  PROC DrawPart12()
    MoveL Offs(pOrigin,202.25,-93.12,-6.00),v60,z5,tcp\WObj:=Plywood;
    MoveL Offs(pOrigin,203.00,-90.38,-6.00),vTravel,z5,tcp\WObj:=Plywood;
    MoveL Offs(pOrigin,203.00,-90.38,-0.00),v60,z0,tcp\WObj:=Plywood;
    MoveL Offs(pOrigin,202.80,-90.22,-0.00),v40,z0,tcp\WObj:=Plywood;
    MoveL Offs(pOrigin,203.15,-89.57,-0.00),v40,z0,tcp\WObj:=Plywood;
    MoveL Offs(pOrigin,202.30,-90.18,-0.00),v40,z0,tcp\WObj:=Plywood;
    MoveL Offs(pOrigin,202.25,-88.72,-0.00),v40,z0,tcp\WObj:=Plywood;
    MoveL Offs(pOrigin,202.60,-88.12,-0.00),v40,z0,tcp\WObj:=Plywood;
    MoveL Offs(pOrigin,202.25,-87.82,-0.00),v40,z0,tcp\WObj:=Plywood;
    MoveL Offs(pOrigin,202.25,-72.22,-0.00),v40,z0,tcp\WObj:=Plywood;
    MoveL Offs(pOrigin,204.35,-70.43,-0.00),v40,z0,tcp\WObj:=Plywood;
    MoveL Offs(pOrigin,203.30,-69.22,-0.00),v40,z0,tcp\WObj:=Plywood;
    MoveL Offs(pOrigin,202.25,-68.93,-0.00),v40,z0,tcp\WObj:=Plywood;
    MoveL Offs(pOrigin,202.10,-50.83,-0.00),v40,z0,tcp\WObj:=Plywood;
    MoveL Offs(pOrigin,210.05,-50.92,-0.00),v40,z0,tcp\WObj:=Plywood;
    MoveL Offs(pOrigin,214.70,-52.12,-0.00),v40,z0,tcp\WObj:=Plywood;
    MoveL Offs(pOrigin,217.55,-53.28,-0.00),v40,z0,tcp\WObj:=Plywood;
    MoveL Offs(pOrigin,222.65,-56.47,-0.00),v40,z0,tcp\WObj:=Plywood;
    MoveL Offs(pOrigin,225.65,-59.33,-0.00),v40,z0,tcp\WObj:=Plywood;
    MoveL Offs(pOrigin,227.75,-62.03,-0.00),v40,z0,tcp\WObj:=Plywood;
    MoveL Offs(pOrigin,229.80,-65.62,-0.00),v40,z0,tcp\WObj:=Plywood;
    MoveL Offs(pOrigin,231.05,-68.78,-0.00),v40,z0,tcp\WObj:=Plywood;
    MoveL Offs(pOrigin,232.25,-74.18,-0.00),v40,z0,tcp\WObj:=Plywood;
    MoveL Offs(pOrigin,232.40,-76.88,-0.00),v40,z0,tcp\WObj:=Plywood;
    MoveL Offs(pOrigin,232.25,-80.93,-0.00),v40,z0,tcp\WObj:=Plywood;
    MoveL Offs(pOrigin,231.50,-84.68,-0.00),v40,z0,tcp\WObj:=Plywood;
    MoveL Offs(pOrigin,230.20,-88.28,-0.00),v40,z0,tcp\WObj:=Plywood;
    MoveL Offs(pOrigin,228.95,-90.38,-0.00),v40,z0,tcp\WObj:=Plywood;
    MoveL Offs(pOrigin,203.00,-90.38,-0.00),v40,z0,tcp\WObj:=Plywood;
    MoveL Offs(pOrigin,203.45,-89.47,-0.00),v40,z0,tcp\WObj:=Plywood;
    MoveL Offs(pOrigin,203.90,-89.32,-0.00),v40,z0,tcp\WObj:=Plywood;
    MoveL Offs(pOrigin,203.45,-88.88,-0.00),v40,z0,tcp\WObj:=Plywood;
    MoveL Offs(pOrigin,203.45,-89.47,-0.00),v40,z0,tcp\WObj:=Plywood;
    MoveL Offs(pOrigin,203.90,-89.18,-0.00),v40,z0,tcp\WObj:=Plywood;
    MoveL Offs(pOrigin,203.60,-88.88,-0.00),v40,z0,tcp\WObj:=Plywood;
    MoveL Offs(pOrigin,203.30,-89.03,-0.00),v40,z0,tcp\WObj:=Plywood;
    MoveL Offs(pOrigin,203.45,-89.47,-0.00),v40,fine,tcp\WObj:=Plywood;
    MoveL Offs(pOrigin,203.45,-89.47,-6.00),v60,z5,tcp\WObj:=Plywood;
    MoveL Offs(pOrigin,198.50,-85.88,-6.00),vTravel,z5,tcp\WObj:=Plywood;
    MoveL Offs(pOrigin,198.50,-85.88,-0.00),v60,z0,tcp\WObj:=Plywood;
    MoveL Offs(pOrigin,198.20,-85.57,-0.00),v40,z0,tcp\WObj:=Plywood;
    MoveL Offs(pOrigin,197.75,-85.88,-0.00),v40,z0,tcp\WObj:=Plywood;
    MoveL Offs(pOrigin,198.35,-86.03,-0.00),v40,z0,tcp\WObj:=Plywood;
    MoveL Offs(pOrigin,198.20,-85.57,-0.00),v40,z0,tcp\WObj:=Plywood;
    MoveL Offs(pOrigin,197.75,-85.88,-0.00),v40,z0,tcp\WObj:=Plywood;
    MoveL Offs(pOrigin,198.50,-85.88,-0.00),v40,z0,tcp\WObj:=Plywood;
    MoveL Offs(pOrigin,197.60,-85.12,-0.00),v40,z0,tcp\WObj:=Plywood;
    MoveL Offs(pOrigin,197.45,-84.32,-0.00),v40,z0,tcp\WObj:=Plywood;
    MoveL Offs(pOrigin,197.15,-84.68,-0.00),v40,z0,tcp\WObj:=Plywood;
    MoveL Offs(pOrigin,197.30,-85.38,-0.00),v40,z0,tcp\WObj:=Plywood;
    MoveL Offs(pOrigin,197.60,-85.12,-0.00),v40,z0,tcp\WObj:=Plywood;
    MoveL Offs(pOrigin,197.65,-84.22,-0.00),v40,z0,tcp\WObj:=Plywood;
    MoveL Offs(pOrigin,199.00,-83.93,-0.00),v40,z0,tcp\WObj:=Plywood;
    MoveL Offs(pOrigin,198.35,-83.53,-0.00),v40,z0,tcp\WObj:=Plywood;
    MoveL Offs(pOrigin,197.65,-84.22,-0.00),v40,fine,tcp\WObj:=Plywood;
    MoveL Offs(pOrigin,197.65,-84.22,-6.00),v60,z5,tcp\WObj:=Plywood;
    MoveL Offs(pOrigin,197.30,-79.53,-6.00),vTravel,z5,tcp\WObj:=Plywood;
    MoveL Offs(pOrigin,197.30,-79.53,-0.00),v60,z0,tcp\WObj:=Plywood;
    MoveL Offs(pOrigin,198.80,-78.38,-0.00),v40,z0,tcp\WObj:=Plywood;
    MoveL Offs(pOrigin,199.10,-77.78,-0.00),v40,z0,tcp\WObj:=Plywood;
    MoveL Offs(pOrigin,199.05,-76.72,-0.00),v40,z0,tcp\WObj:=Plywood;
    MoveL Offs(pOrigin,197.90,-75.82,-0.00),v40,z0,tcp\WObj:=Plywood;
    MoveL Offs(pOrigin,197.50,-76.28,-0.00),v40,z0,tcp\WObj:=Plywood;
    MoveL Offs(pOrigin,198.40,-76.88,-0.00),v40,z0,tcp\WObj:=Plywood;
    MoveL Offs(pOrigin,198.50,-77.32,-0.00),v40,z0,tcp\WObj:=Plywood;
    MoveL Offs(pOrigin,197.15,-76.57,-0.00),v40,z0,tcp\WObj:=Plywood;
    MoveL Offs(pOrigin,196.40,-77.03,-0.00),v40,z0,tcp\WObj:=Plywood;
    MoveL Offs(pOrigin,195.80,-77.93,-0.00),v40,z0,tcp\WObj:=Plywood;
    MoveL Offs(pOrigin,195.90,-78.68,-0.00),v40,z0,tcp\WObj:=Plywood;
    MoveL Offs(pOrigin,196.85,-79.53,-0.00),v40,z0,tcp\WObj:=Plywood;
    MoveL Offs(pOrigin,197.30,-79.53,-0.00),v40,z0,tcp\WObj:=Plywood;
    MoveL Offs(pOrigin,196.85,-78.78,-0.00),v40,z0,tcp\WObj:=Plywood;
    MoveL Offs(pOrigin,196.65,-77.93,-0.00),v40,z0,tcp\WObj:=Plywood;
    MoveL Offs(pOrigin,197.45,-77.38,-0.00),v40,z0,tcp\WObj:=Plywood;
    MoveL Offs(pOrigin,197.65,-78.22,-0.00),v40,z0,tcp\WObj:=Plywood;
    MoveL Offs(pOrigin,196.85,-78.78,-0.00),v40,fine,tcp\WObj:=Plywood;
    MoveL Offs(pOrigin,196.85,-78.78,-6.00),v60,z5,tcp\WObj:=Plywood;
    MoveL Offs(pOrigin,195.80,-77.32,-6.00),vTravel,z5,tcp\WObj:=Plywood;
    MoveL Offs(pOrigin,195.80,-77.32,-0.00),v60,z0,tcp\WObj:=Plywood;
    MoveL Offs(pOrigin,196.90,-75.97,-0.00),v40,z0,tcp\WObj:=Plywood;
    MoveL Offs(pOrigin,196.55,-75.68,-0.00),v40,z0,tcp\WObj:=Plywood;
    MoveL Offs(pOrigin,195.35,-76.72,-0.00),v40,z0,tcp\WObj:=Plywood;
    MoveL Offs(pOrigin,194.80,-76.57,-0.00),v40,z0,tcp\WObj:=Plywood;
    MoveL Offs(pOrigin,194.80,-76.12,-0.00),v40,z0,tcp\WObj:=Plywood;
    MoveL Offs(pOrigin,195.95,-74.78,-0.00),v40,z0,tcp\WObj:=Plywood;
    MoveL Offs(pOrigin,195.65,-74.43,-0.00),v40,z0,tcp\WObj:=Plywood;
    MoveL Offs(pOrigin,194.90,-74.62,-0.00),v40,z0,tcp\WObj:=Plywood;
    MoveL Offs(pOrigin,195.00,-73.88,-0.00),v40,z0,tcp\WObj:=Plywood;
    MoveL Offs(pOrigin,194.35,-73.12,-0.00),v40,z0,tcp\WObj:=Plywood;
    MoveL Offs(pOrigin,194.60,-72.07,-0.00),v40,z0,tcp\WObj:=Plywood;
    MoveL Offs(pOrigin,194.15,-71.82,-0.00),v40,z0,tcp\WObj:=Plywood;
    MoveL Offs(pOrigin,192.85,-73.07,-0.00),v40,z0,tcp\WObj:=Plywood;
    MoveL Offs(pOrigin,193.30,-72.22,-0.00),v40,z0,tcp\WObj:=Plywood;
    MoveL Offs(pOrigin,192.80,-71.93,-0.00),v40,z0,tcp\WObj:=Plywood;
    MoveL Offs(pOrigin,191.45,-72.97,-0.00),v40,z0,tcp\WObj:=Plywood;
    MoveL Offs(pOrigin,191.25,-72.22,-0.00),v40,z0,tcp\WObj:=Plywood;
    MoveL Offs(pOrigin,192.20,-71.03,-0.00),v40,z0,tcp\WObj:=Plywood;
    MoveL Offs(pOrigin,191.75,-70.72,-0.00),v40,z0,tcp\WObj:=Plywood;
    MoveL Offs(pOrigin,191.00,-71.07,-0.00),v40,z0,tcp\WObj:=Plywood;
    MoveL Offs(pOrigin,189.85,-72.38,-0.00),v40,z0,tcp\WObj:=Plywood;
    MoveL Offs(pOrigin,189.95,-72.82,-0.00),v40,z0,tcp\WObj:=Plywood;
    MoveL Offs(pOrigin,191.00,-73.88,-0.00),v40,z0,tcp\WObj:=Plywood;
    MoveL Offs(pOrigin,191.75,-73.88,-0.00),v40,z0,tcp\WObj:=Plywood;
    MoveL Offs(pOrigin,192.35,-73.43,-0.00),v40,z0,tcp\WObj:=Plywood;
    MoveL Offs(pOrigin,191.75,-74.47,-0.00),v40,z0,tcp\WObj:=Plywood;
    MoveL Offs(pOrigin,192.50,-75.53,-0.00),v40,z0,tcp\WObj:=Plywood;
    MoveL Offs(pOrigin,193.95,-75.72,-0.00),v40,z0,tcp\WObj:=Plywood;
    MoveL Offs(pOrigin,193.75,-76.43,-0.00),v40,z0,tcp\WObj:=Plywood;
    MoveL Offs(pOrigin,194.75,-77.57,-0.00),v40,z0,tcp\WObj:=Plywood;
    MoveL Offs(pOrigin,195.80,-77.32,-0.00),v40,fine,tcp\WObj:=Plywood;
    MoveL Offs(pOrigin,195.80,-77.32,-6.00),v60,z5,tcp\WObj:=Plywood;
    MoveL Offs(pOrigin,193.85,-74.72,-6.00),vTravel,z5,tcp\WObj:=Plywood;
    MoveL Offs(pOrigin,193.85,-74.72,-0.00),v60,z0,tcp\WObj:=Plywood;
    MoveL Offs(pOrigin,193.00,-74.78,-0.00),v40,z0,tcp\WObj:=Plywood;
    MoveL Offs(pOrigin,193.25,-74.03,-0.00),v40,z0,tcp\WObj:=Plywood;
    MoveL Offs(pOrigin,194.00,-73.88,-0.00),v40,z0,tcp\WObj:=Plywood;
    MoveL Offs(pOrigin,193.85,-74.72,-0.00),v40,fine,tcp\WObj:=Plywood;
    MoveL Offs(pOrigin,193.85,-74.72,-6.00),v60,z5,tcp\WObj:=Plywood;
    MoveL Offs(pOrigin,191.40,-70.57,-6.00),vTravel,z5,tcp\WObj:=Plywood;
    MoveL Offs(pOrigin,191.40,-70.57,-0.00),v60,z0,tcp\WObj:=Plywood;
  ENDPROC

  PROC DrawPart13()
    MoveL Offs(pOrigin,190.55,-69.38,-0.00),v40,z0,tcp\WObj:=Plywood;
    MoveL Offs(pOrigin,189.80,-68.93,-0.00),v40,z0,tcp\WObj:=Plywood;
    MoveL Offs(pOrigin,188.95,-69.68,-0.00),v40,z0,tcp\WObj:=Plywood;
    MoveL Offs(pOrigin,189.45,-71.12,-0.00),v40,z0,tcp\WObj:=Plywood;
    MoveL Offs(pOrigin,188.75,-70.18,-0.00),v40,z0,tcp\WObj:=Plywood;
    MoveL Offs(pOrigin,188.30,-70.43,-0.00),v40,z0,tcp\WObj:=Plywood;
    MoveL Offs(pOrigin,188.60,-71.47,-0.00),v40,z0,tcp\WObj:=Plywood;
    MoveL Offs(pOrigin,189.35,-71.93,-0.00),v40,z0,tcp\WObj:=Plywood;
    MoveL Offs(pOrigin,189.95,-71.88,-0.00),v40,z0,tcp\WObj:=Plywood;
    MoveL Offs(pOrigin,191.40,-70.57,-0.00),v40,fine,tcp\WObj:=Plywood;
    MoveL Offs(pOrigin,191.40,-70.57,-6.00),v60,z5,tcp\WObj:=Plywood;
    MoveL Offs(pOrigin,190.10,-70.43,-6.00),vTravel,z5,tcp\WObj:=Plywood;
    MoveL Offs(pOrigin,190.10,-70.43,-0.00),v60,z0,tcp\WObj:=Plywood;
    MoveL Offs(pOrigin,189.80,-69.82,-0.00),v40,z0,tcp\WObj:=Plywood;
    MoveL Offs(pOrigin,190.10,-70.43,-0.00),v40,fine,tcp\WObj:=Plywood;
    MoveL Offs(pOrigin,190.10,-70.43,-6.00),v60,z5,tcp\WObj:=Plywood;
    MoveL Offs(pOrigin,188.65,-69.38,-6.00),vTravel,z5,tcp\WObj:=Plywood;
    MoveL Offs(pOrigin,188.65,-69.38,-0.00),v60,z0,tcp\WObj:=Plywood;
    MoveL Offs(pOrigin,187.70,-67.93,-0.00),v40,z0,tcp\WObj:=Plywood;
    MoveL Offs(pOrigin,188.45,-68.18,-0.00),v40,z0,tcp\WObj:=Plywood;
    MoveL Offs(pOrigin,188.75,-69.03,-0.00),v40,z0,tcp\WObj:=Plywood;
    MoveL Offs(pOrigin,189.15,-68.78,-0.00),v40,z0,tcp\WObj:=Plywood;
    MoveL Offs(pOrigin,189.10,-68.18,-0.00),v40,z0,tcp\WObj:=Plywood;
    MoveL Offs(pOrigin,188.45,-67.47,-0.00),v40,z0,tcp\WObj:=Plywood;
    MoveL Offs(pOrigin,187.40,-67.47,-0.00),v40,z0,tcp\WObj:=Plywood;
    MoveL Offs(pOrigin,186.70,-68.18,-0.00),v40,z0,tcp\WObj:=Plywood;
    MoveL Offs(pOrigin,186.50,-68.78,-0.00),v40,z0,tcp\WObj:=Plywood;
    MoveL Offs(pOrigin,187.25,-69.93,-0.00),v40,z0,tcp\WObj:=Plywood;
    MoveL Offs(pOrigin,188.15,-69.88,-0.00),v40,z0,tcp\WObj:=Plywood;
    MoveL Offs(pOrigin,188.65,-69.38,-0.00),v40,z0,tcp\WObj:=Plywood;
    MoveL Offs(pOrigin,187.80,-69.22,-0.00),v40,z0,tcp\WObj:=Plywood;
    MoveL Offs(pOrigin,187.25,-69.18,-0.00),v40,z0,tcp\WObj:=Plywood;
    MoveL Offs(pOrigin,187.15,-68.68,-0.00),v40,z0,tcp\WObj:=Plywood;
    MoveL Offs(pOrigin,187.80,-69.22,-0.00),v40,fine,tcp\WObj:=Plywood;
    MoveL Offs(pOrigin,187.80,-69.22,-6.00),v60,z5,tcp\WObj:=Plywood;
    MoveL Offs(pOrigin,186.45,-67.88,-6.00),vTravel,z5,tcp\WObj:=Plywood;
    MoveL Offs(pOrigin,186.45,-67.88,-0.00),v60,z0,tcp\WObj:=Plywood;
    MoveL Offs(pOrigin,187.35,-66.82,-0.00),v40,z0,tcp\WObj:=Plywood;
    MoveL Offs(pOrigin,187.25,-66.57,-0.00),v40,z0,tcp\WObj:=Plywood;
    MoveL Offs(pOrigin,185.45,-68.18,-0.00),v40,z0,tcp\WObj:=Plywood;
    MoveL Offs(pOrigin,185.20,-68.78,-0.00),v40,z0,tcp\WObj:=Plywood;
    MoveL Offs(pOrigin,186.45,-67.88,-0.00),v40,fine,tcp\WObj:=Plywood;
    MoveL Offs(pOrigin,186.45,-67.88,-6.00),v60,z5,tcp\WObj:=Plywood;
    MoveL Offs(pOrigin,186.50,-66.38,-6.00),vTravel,z5,tcp\WObj:=Plywood;
    MoveL Offs(pOrigin,186.50,-66.38,-0.00),v60,z0,tcp\WObj:=Plywood;
    MoveL Offs(pOrigin,186.50,-65.62,-0.00),v40,z0,tcp\WObj:=Plywood;
    MoveL Offs(pOrigin,186.50,-66.38,-0.00),v40,fine,tcp\WObj:=Plywood;
    MoveL Offs(pOrigin,186.50,-66.38,-6.00),v60,z5,tcp\WObj:=Plywood;
    MoveL Offs(pOrigin,185.30,-76.07,-6.00),vTravel,z5,tcp\WObj:=Plywood;
    MoveL Offs(pOrigin,185.30,-76.07,-0.00),v60,z0,tcp\WObj:=Plywood;
    MoveL Offs(pOrigin,185.05,-76.28,-0.00),v40,z0,tcp\WObj:=Plywood;
    MoveL Offs(pOrigin,185.75,-77.32,-0.00),v40,z0,tcp\WObj:=Plywood;
    MoveL Offs(pOrigin,185.05,-77.47,-0.00),v40,z0,tcp\WObj:=Plywood;
    MoveL Offs(pOrigin,185.00,-78.62,-0.00),v40,z0,tcp\WObj:=Plywood;
    MoveL Offs(pOrigin,186.25,-77.32,-0.00),v40,z0,tcp\WObj:=Plywood;
    MoveL Offs(pOrigin,185.30,-76.07,-0.00),v40,fine,tcp\WObj:=Plywood;
    MoveL Offs(pOrigin,185.30,-76.07,-6.00),v60,z5,tcp\WObj:=Plywood;
    MoveL Offs(pOrigin,184.05,-77.03,-6.00),vTravel,z5,tcp\WObj:=Plywood;
    MoveL Offs(pOrigin,184.05,-77.03,-0.00),v60,z0,tcp\WObj:=Plywood;
    MoveL Offs(pOrigin,184.75,-77.03,-0.00),v40,z0,tcp\WObj:=Plywood;
    MoveL Offs(pOrigin,184.05,-77.03,-0.00),v40,fine,tcp\WObj:=Plywood;
    MoveL Offs(pOrigin,184.05,-77.03,-6.00),v60,z5,tcp\WObj:=Plywood;
    MoveL Offs(pOrigin,184.95,-78.68,-6.00),vTravel,z5,tcp\WObj:=Plywood;
    MoveL Offs(pOrigin,184.95,-78.68,-0.00),v60,z0,tcp\WObj:=Plywood;
    MoveL Offs(pOrigin,184.10,-78.97,-0.00),v40,z0,tcp\WObj:=Plywood;
    MoveL Offs(pOrigin,184.10,-79.28,-0.00),v40,z0,tcp\WObj:=Plywood;
    MoveL Offs(pOrigin,184.70,-79.12,-0.00),v40,z0,tcp\WObj:=Plywood;
    MoveL Offs(pOrigin,184.95,-78.68,-0.00),v40,fine,tcp\WObj:=Plywood;
    MoveL Offs(pOrigin,184.95,-78.68,-6.00),v60,z5,tcp\WObj:=Plywood;
    MoveL Offs(pOrigin,197.15,-66.68,-6.00),vTravel,z5,tcp\WObj:=Plywood;
    MoveL Offs(pOrigin,197.15,-66.68,-0.00),v60,z0,tcp\WObj:=Plywood;
    MoveL Offs(pOrigin,197.90,-67.38,-0.00),v40,z0,tcp\WObj:=Plywood;
    MoveL Offs(pOrigin,198.50,-67.38,-0.00),v40,z0,tcp\WObj:=Plywood;
    MoveL Offs(pOrigin,198.60,-66.97,-0.00),v40,z0,tcp\WObj:=Plywood;
    MoveL Offs(pOrigin,197.80,-66.62,-0.00),v40,z0,tcp\WObj:=Plywood;
    MoveL Offs(pOrigin,197.55,-65.62,-0.00),v40,z0,tcp\WObj:=Plywood;
    MoveL Offs(pOrigin,197.30,-65.62,-0.00),v40,z0,tcp\WObj:=Plywood;
    MoveL Offs(pOrigin,197.00,-66.07,-0.00),v40,z0,tcp\WObj:=Plywood;
    MoveL Offs(pOrigin,197.15,-66.68,-0.00),v40,fine,tcp\WObj:=Plywood;
    MoveL Offs(pOrigin,197.15,-66.68,-6.00),v60,z5,tcp\WObj:=Plywood;
    MoveL Offs(pOrigin,197.65,-65.47,-6.00),vTravel,z5,tcp\WObj:=Plywood;
    MoveL Offs(pOrigin,197.65,-65.47,-0.00),v60,z0,tcp\WObj:=Plywood;
    MoveL Offs(pOrigin,199.00,-65.18,-0.00),v40,z0,tcp\WObj:=Plywood;
    MoveL Offs(pOrigin,198.20,-64.88,-0.00),v40,z0,tcp\WObj:=Plywood;
    MoveL Offs(pOrigin,197.65,-65.47,-0.00),v40,fine,tcp\WObj:=Plywood;
    MoveL Offs(pOrigin,197.65,-65.47,-6.00),v60,z5,tcp\WObj:=Plywood;
    MoveL Offs(pOrigin,202.70,-69.68,-6.00),vTravel,z5,tcp\WObj:=Plywood;
    MoveL Offs(pOrigin,202.70,-69.68,-0.00),v60,z0,tcp\WObj:=Plywood;
    MoveL Offs(pOrigin,203.00,-69.97,-0.00),v40,z0,tcp\WObj:=Plywood;
    MoveL Offs(pOrigin,202.85,-70.43,-0.00),v40,z0,tcp\WObj:=Plywood;
    MoveL Offs(pOrigin,202.70,-69.68,-0.00),v40,z0,tcp\WObj:=Plywood;
    MoveL Offs(pOrigin,203.00,-69.97,-0.00),v40,z0,tcp\WObj:=Plywood;
    MoveL Offs(pOrigin,202.85,-70.43,-0.00),v40,z0,tcp\WObj:=Plywood;
    MoveL Offs(pOrigin,202.70,-69.68,-0.00),v40,fine,tcp\WObj:=Plywood;
    MoveL Offs(pOrigin,202.70,-69.68,-6.00),v60,z5,tcp\WObj:=Plywood;
    MoveL Offs(pOrigin,204.65,-70.72,-6.00),vTravel,z5,tcp\WObj:=Plywood;
    MoveL Offs(pOrigin,204.65,-70.72,-0.00),v60,z0,tcp\WObj:=Plywood;
    MoveL Offs(pOrigin,202.85,-72.38,-0.00),v40,z0,tcp\WObj:=Plywood;
    MoveL Offs(pOrigin,203.00,-72.97,-0.00),v40,z0,tcp\WObj:=Plywood;
    MoveL Offs(pOrigin,204.05,-73.88,-0.00),v40,z0,tcp\WObj:=Plywood;
    MoveL Offs(pOrigin,204.95,-73.72,-0.00),v40,z0,tcp\WObj:=Plywood;
    MoveL Offs(pOrigin,206.25,-72.38,-0.00),v40,z0,tcp\WObj:=Plywood;
    MoveL Offs(pOrigin,205.70,-71.82,-0.00),v40,z0,tcp\WObj:=Plywood;
    MoveL Offs(pOrigin,204.35,-72.93,-0.00),v40,z0,tcp\WObj:=Plywood;
    MoveL Offs(pOrigin,204.10,-72.82,-0.00),v40,z0,tcp\WObj:=Plywood;
    MoveL Offs(pOrigin,204.10,-72.38,-0.00),v40,z0,tcp\WObj:=Plywood;
    MoveL Offs(pOrigin,205.10,-71.18,-0.00),v40,z0,tcp\WObj:=Plywood;
    MoveL Offs(pOrigin,204.65,-70.72,-0.00),v40,fine,tcp\WObj:=Plywood;
    MoveL Offs(pOrigin,204.65,-70.72,-6.00),v60,z5,tcp\WObj:=Plywood;
    MoveL Offs(pOrigin,206.75,-72.12,-6.00),vTravel,z5,tcp\WObj:=Plywood;
    MoveL Offs(pOrigin,206.75,-72.12,-0.00),v60,z0,tcp\WObj:=Plywood;
    MoveL Offs(pOrigin,204.85,-73.88,-0.00),v40,z0,tcp\WObj:=Plywood;
    MoveL Offs(pOrigin,204.70,-74.62,-0.00),v40,z0,tcp\WObj:=Plywood;
    MoveL Offs(pOrigin,205.85,-75.78,-0.00),v40,z0,tcp\WObj:=Plywood;
    MoveL Offs(pOrigin,206.65,-75.88,-0.00),v40,z0,tcp\WObj:=Plywood;
    MoveL Offs(pOrigin,206.50,-76.43,-0.00),v40,z0,tcp\WObj:=Plywood;
    MoveL Offs(pOrigin,207.50,-77.47,-0.00),v40,z0,tcp\WObj:=Plywood;
    MoveL Offs(pOrigin,208.80,-77.43,-0.00),v40,z0,tcp\WObj:=Plywood;
    MoveL Offs(pOrigin,208.55,-78.22,-0.00),v40,z0,tcp\WObj:=Plywood;
    MoveL Offs(pOrigin,208.75,-78.82,-0.00),v40,z0,tcp\WObj:=Plywood;
  ENDPROC

  PROC DrawPart14()
    MoveL Offs(pOrigin,209.90,-79.68,-0.00),v40,z0,tcp\WObj:=Plywood;
    MoveL Offs(pOrigin,210.35,-79.62,-0.00),v40,z0,tcp\WObj:=Plywood;
    MoveL Offs(pOrigin,212.10,-77.93,-0.00),v40,z0,tcp\WObj:=Plywood;
    MoveL Offs(pOrigin,212.30,-76.43,-0.00),v40,z0,tcp\WObj:=Plywood;
    MoveL Offs(pOrigin,211.45,-75.78,-0.00),v40,z0,tcp\WObj:=Plywood;
    MoveL Offs(pOrigin,211.40,-75.22,-0.00),v40,z0,tcp\WObj:=Plywood;
    MoveL Offs(pOrigin,212.15,-75.57,-0.00),v40,z0,tcp\WObj:=Plywood;
    MoveL Offs(pOrigin,212.70,-75.07,-0.00),v40,z0,tcp\WObj:=Plywood;
    MoveL Offs(pOrigin,212.70,-72.97,-0.00),v40,z0,tcp\WObj:=Plywood;
    MoveL Offs(pOrigin,212.15,-72.68,-0.00),v40,z0,tcp\WObj:=Plywood;
    MoveL Offs(pOrigin,210.65,-72.68,-0.00),v40,z0,tcp\WObj:=Plywood;
    MoveL Offs(pOrigin,210.20,-72.12,-0.00),v40,z0,tcp\WObj:=Plywood;
    MoveL Offs(pOrigin,209.85,-72.78,-0.00),v40,z0,tcp\WObj:=Plywood;
    MoveL Offs(pOrigin,208.90,-72.97,-0.00),v40,z0,tcp\WObj:=Plywood;
    MoveL Offs(pOrigin,209.85,-73.43,-0.00),v40,z0,tcp\WObj:=Plywood;
    MoveL Offs(pOrigin,209.75,-74.78,-0.00),v40,z0,tcp\WObj:=Plywood;
    MoveL Offs(pOrigin,210.20,-75.97,-0.00),v40,z0,tcp\WObj:=Plywood;
    MoveL Offs(pOrigin,209.60,-75.53,-0.00),v40,z0,tcp\WObj:=Plywood;
    MoveL Offs(pOrigin,208.05,-75.88,-0.00),v40,z0,tcp\WObj:=Plywood;
    MoveL Offs(pOrigin,208.40,-75.43,-0.00),v40,z0,tcp\WObj:=Plywood;
    MoveL Offs(pOrigin,209.60,-75.32,-0.00),v40,z0,tcp\WObj:=Plywood;
    MoveL Offs(pOrigin,209.75,-74.93,-0.00),v40,z0,tcp\WObj:=Plywood;
    MoveL Offs(pOrigin,208.55,-74.18,-0.00),v40,z0,tcp\WObj:=Plywood;
    MoveL Offs(pOrigin,208.10,-74.22,-0.00),v40,z0,tcp\WObj:=Plywood;
    MoveL Offs(pOrigin,207.85,-74.68,-0.00),v40,z0,tcp\WObj:=Plywood;
    MoveL Offs(pOrigin,208.05,-73.72,-0.00),v40,z0,tcp\WObj:=Plywood;
    MoveL Offs(pOrigin,208.65,-72.97,-0.00),v40,z0,tcp\WObj:=Plywood;
    MoveL Offs(pOrigin,207.80,-72.72,-0.00),v40,z0,tcp\WObj:=Plywood;
    MoveL Offs(pOrigin,207.35,-72.12,-0.00),v40,z0,tcp\WObj:=Plywood;
    MoveL Offs(pOrigin,206.75,-72.12,-0.00),v40,fine,tcp\WObj:=Plywood;
    MoveL Offs(pOrigin,206.75,-72.12,-6.00),v60,z5,tcp\WObj:=Plywood;
    MoveL Offs(pOrigin,206.30,-73.93,-6.00),vTravel,z5,tcp\WObj:=Plywood;
    MoveL Offs(pOrigin,206.30,-73.93,-0.00),v60,z0,tcp\WObj:=Plywood;
    MoveL Offs(pOrigin,207.00,-74.18,-0.00),v40,z0,tcp\WObj:=Plywood;
    MoveL Offs(pOrigin,206.60,-74.82,-0.00),v40,z0,tcp\WObj:=Plywood;
    MoveL Offs(pOrigin,205.90,-74.78,-0.00),v40,z0,tcp\WObj:=Plywood;
    MoveL Offs(pOrigin,206.30,-73.93,-0.00),v40,z0,tcp\WObj:=Plywood;
    MoveL Offs(pOrigin,206.30,-74.32,-0.00),v40,z0,tcp\WObj:=Plywood;
    MoveL Offs(pOrigin,206.15,-74.62,-0.00),v40,z0,tcp\WObj:=Plywood;
    MoveL Offs(pOrigin,206.60,-74.62,-0.00),v40,z0,tcp\WObj:=Plywood;
    MoveL Offs(pOrigin,206.45,-74.32,-0.00),v40,z0,tcp\WObj:=Plywood;
    MoveL Offs(pOrigin,206.15,-74.62,-0.00),v40,z0,tcp\WObj:=Plywood;
    MoveL Offs(pOrigin,206.45,-74.78,-0.00),v40,z0,tcp\WObj:=Plywood;
    MoveL Offs(pOrigin,206.60,-74.47,-0.00),v40,z0,tcp\WObj:=Plywood;
    MoveL Offs(pOrigin,206.30,-74.32,-0.00),v40,fine,tcp\WObj:=Plywood;
    MoveL Offs(pOrigin,206.30,-74.32,-6.00),v60,z5,tcp\WObj:=Plywood;
    MoveL Offs(pOrigin,208.85,-73.88,-6.00),vTravel,z5,tcp\WObj:=Plywood;
    MoveL Offs(pOrigin,208.85,-73.88,-0.00),v60,z0,tcp\WObj:=Plywood;
    MoveL Offs(pOrigin,209.45,-73.88,-0.00),v40,z0,tcp\WObj:=Plywood;
    MoveL Offs(pOrigin,208.85,-73.88,-0.00),v40,fine,tcp\WObj:=Plywood;
    MoveL Offs(pOrigin,208.85,-73.88,-6.00),v60,z5,tcp\WObj:=Plywood;
    MoveL Offs(pOrigin,210.35,-77.53,-6.00),vTravel,z5,tcp\WObj:=Plywood;
    MoveL Offs(pOrigin,210.35,-77.53,-0.00),v60,z0,tcp\WObj:=Plywood;
    MoveL Offs(pOrigin,210.40,-78.22,-0.00),v40,z0,tcp\WObj:=Plywood;
    MoveL Offs(pOrigin,209.85,-78.53,-0.00),v40,z0,tcp\WObj:=Plywood;
    MoveL Offs(pOrigin,210.05,-78.22,-0.00),v40,z0,tcp\WObj:=Plywood;
    MoveL Offs(pOrigin,209.65,-77.78,-0.00),v40,z0,tcp\WObj:=Plywood;
    MoveL Offs(pOrigin,210.35,-77.53,-0.00),v40,fine,tcp\WObj:=Plywood;
    MoveL Offs(pOrigin,210.35,-77.53,-6.00),v60,z5,tcp\WObj:=Plywood;
    MoveL Offs(pOrigin,210.95,-83.57,-6.00),vTravel,z5,tcp\WObj:=Plywood;
    MoveL Offs(pOrigin,210.95,-83.57,-0.00),v60,z0,tcp\WObj:=Plywood;
    MoveL Offs(pOrigin,209.95,-84.68,-0.00),v40,z0,tcp\WObj:=Plywood;
    MoveL Offs(pOrigin,210.65,-85.93,-0.00),v40,z0,tcp\WObj:=Plywood;
    MoveL Offs(pOrigin,211.30,-85.88,-0.00),v40,z0,tcp\WObj:=Plywood;
    MoveL Offs(pOrigin,210.50,-85.12,-0.00),v40,z0,tcp\WObj:=Plywood;
    MoveL Offs(pOrigin,211.10,-84.18,-0.00),v40,z0,tcp\WObj:=Plywood;
    MoveL Offs(pOrigin,211.70,-84.18,-0.00),v40,z0,tcp\WObj:=Plywood;
    MoveL Offs(pOrigin,212.40,-84.97,-0.00),v40,z0,tcp\WObj:=Plywood;
    MoveL Offs(pOrigin,212.40,-84.22,-0.00),v40,z0,tcp\WObj:=Plywood;
    MoveL Offs(pOrigin,211.70,-83.53,-0.00),v40,z0,tcp\WObj:=Plywood;
    MoveL Offs(pOrigin,210.95,-83.57,-0.00),v40,fine,tcp\WObj:=Plywood;
    MoveL Offs(pOrigin,210.95,-83.57,-6.00),v60,z5,tcp\WObj:=Plywood;
    MoveL Offs(pOrigin,212.75,-85.43,-6.00),vTravel,z5,tcp\WObj:=Plywood;
    MoveL Offs(pOrigin,212.75,-85.43,-0.00),v60,z0,tcp\WObj:=Plywood;
    MoveL Offs(pOrigin,211.00,-87.38,-0.00),v40,z0,tcp\WObj:=Plywood;
    MoveL Offs(pOrigin,211.40,-87.32,-0.00),v40,z0,tcp\WObj:=Plywood;
    MoveL Offs(pOrigin,213.15,-85.43,-0.00),v40,z0,tcp\WObj:=Plywood;
    MoveL Offs(pOrigin,212.75,-85.43,-0.00),v40,z0,tcp\WObj:=Plywood;
    MoveL Offs(pOrigin,213.05,-86.47,-0.00),v40,z0,tcp\WObj:=Plywood;
    MoveL Offs(pOrigin,212.60,-86.93,-0.00),v40,z0,tcp\WObj:=Plywood;
    MoveL Offs(pOrigin,213.05,-87.07,-0.00),v40,z0,tcp\WObj:=Plywood;
    MoveL Offs(pOrigin,213.20,-86.47,-0.00),v40,z0,tcp\WObj:=Plywood;
    MoveL Offs(pOrigin,212.60,-86.93,-0.00),v40,z0,tcp\WObj:=Plywood;
    MoveL Offs(pOrigin,213.05,-87.07,-0.00),v40,z0,tcp\WObj:=Plywood;
    MoveL Offs(pOrigin,213.35,-86.62,-0.00),v40,z0,tcp\WObj:=Plywood;
    MoveL Offs(pOrigin,213.05,-86.47,-0.00),v40,fine,tcp\WObj:=Plywood;
    MoveL Offs(pOrigin,213.05,-86.47,-6.00),v60,z5,tcp\WObj:=Plywood;
    MoveL Offs(pOrigin,219.70,-76.28,-6.00),vTravel,z5,tcp\WObj:=Plywood;
    MoveL Offs(pOrigin,219.70,-76.28,-0.00),v60,z0,tcp\WObj:=Plywood;
    MoveL Offs(pOrigin,220.20,-76.43,-0.00),v40,z0,tcp\WObj:=Plywood;
    MoveL Offs(pOrigin,220.65,-75.53,-0.00),v40,z0,tcp\WObj:=Plywood;
    MoveL Offs(pOrigin,220.10,-75.68,-0.00),v40,z0,tcp\WObj:=Plywood;
    MoveL Offs(pOrigin,219.70,-76.28,-0.00),v40,z0,tcp\WObj:=Plywood;
    MoveL Offs(pOrigin,219.65,-75.53,-0.00),v40,z0,tcp\WObj:=Plywood;
    MoveL Offs(pOrigin,220.45,-74.62,-0.00),v40,z0,tcp\WObj:=Plywood;
    MoveL Offs(pOrigin,220.25,-74.38,-0.00),v40,z0,tcp\WObj:=Plywood;
    MoveL Offs(pOrigin,219.50,-75.07,-0.00),v40,z0,tcp\WObj:=Plywood;
    MoveL Offs(pOrigin,218.90,-75.03,-0.00),v40,z0,tcp\WObj:=Plywood;
    MoveL Offs(pOrigin,218.60,-74.62,-0.00),v40,z0,tcp\WObj:=Plywood;
    MoveL Offs(pOrigin,219.95,-72.43,-0.00),v40,z0,tcp\WObj:=Plywood;
    MoveL Offs(pOrigin,217.70,-74.32,-0.00),v40,z0,tcp\WObj:=Plywood;
    MoveL Offs(pOrigin,218.45,-75.38,-0.00),v40,z0,tcp\WObj:=Plywood;
    MoveL Offs(pOrigin,219.05,-75.68,-0.00),v40,z0,tcp\WObj:=Plywood;
    MoveL Offs(pOrigin,219.65,-75.53,-0.00),v40,fine,tcp\WObj:=Plywood;
    MoveL Offs(pOrigin,219.65,-75.53,-6.00),v60,z5,tcp\WObj:=Plywood;
    MoveL Offs(pOrigin,217.10,-73.82,-6.00),vTravel,z5,tcp\WObj:=Plywood;
    MoveL Offs(pOrigin,217.10,-73.82,-0.00),v60,z0,tcp\WObj:=Plywood;
    MoveL Offs(pOrigin,218.75,-72.38,-0.00),v40,z0,tcp\WObj:=Plywood;
    MoveL Offs(pOrigin,218.45,-72.12,-0.00),v40,z0,tcp\WObj:=Plywood;
    MoveL Offs(pOrigin,217.25,-73.07,-0.00),v40,z0,tcp\WObj:=Plywood;
    MoveL Offs(pOrigin,216.85,-72.97,-0.00),v40,z0,tcp\WObj:=Plywood;
    MoveL Offs(pOrigin,216.75,-72.38,-0.00),v40,z0,tcp\WObj:=Plywood;
    MoveL Offs(pOrigin,217.65,-71.32,-0.00),v40,z0,tcp\WObj:=Plywood;
    MoveL Offs(pOrigin,217.55,-70.93,-0.00),v40,z0,tcp\WObj:=Plywood;
    MoveL Offs(pOrigin,216.95,-71.18,-0.00),v40,z0,tcp\WObj:=Plywood;
    MoveL Offs(pOrigin,215.75,-72.53,-0.00),v40,z0,tcp\WObj:=Plywood;
    MoveL Offs(pOrigin,216.50,-73.57,-0.00),v40,z0,tcp\WObj:=Plywood;
    MoveL Offs(pOrigin,217.10,-73.82,-0.00),v40,fine,tcp\WObj:=Plywood;
    MoveL Offs(pOrigin,217.10,-73.82,-6.00),v60,z5,tcp\WObj:=Plywood;
    MoveL Offs(pOrigin,215.90,-71.62,-6.00),vTravel,z5,tcp\WObj:=Plywood;
  ENDPROC

  PROC DrawPart15()
    MoveL Offs(pOrigin,215.90,-71.62,-0.00),v60,z0,tcp\WObj:=Plywood;
    MoveL Offs(pOrigin,216.95,-70.43,-0.00),v40,z0,tcp\WObj:=Plywood;
    MoveL Offs(pOrigin,216.20,-69.38,-0.00),v40,z0,tcp\WObj:=Plywood;
    MoveL Offs(pOrigin,215.60,-69.07,-0.00),v40,z0,tcp\WObj:=Plywood;
    MoveL Offs(pOrigin,214.70,-69.68,-0.00),v40,z0,tcp\WObj:=Plywood;
    MoveL Offs(pOrigin,215.10,-71.12,-0.00),v40,z0,tcp\WObj:=Plywood;
    MoveL Offs(pOrigin,214.55,-70.12,-0.00),v40,z0,tcp\WObj:=Plywood;
    MoveL Offs(pOrigin,214.25,-70.12,-0.00),v40,z0,tcp\WObj:=Plywood;
    MoveL Offs(pOrigin,214.00,-70.72,-0.00),v40,z0,tcp\WObj:=Plywood;
    MoveL Offs(pOrigin,214.40,-71.62,-0.00),v40,z0,tcp\WObj:=Plywood;
    MoveL Offs(pOrigin,215.00,-72.03,-0.00),v40,z0,tcp\WObj:=Plywood;
    MoveL Offs(pOrigin,215.90,-71.62,-0.00),v40,z0,tcp\WObj:=Plywood;
    MoveL Offs(pOrigin,215.90,-70.47,-0.00),v40,z0,tcp\WObj:=Plywood;
    MoveL Offs(pOrigin,215.45,-69.97,-0.00),v40,z0,tcp\WObj:=Plywood;
    MoveL Offs(pOrigin,215.75,-69.68,-0.00),v40,z0,tcp\WObj:=Plywood;
    MoveL Offs(pOrigin,216.05,-70.12,-0.00),v40,z0,tcp\WObj:=Plywood;
    MoveL Offs(pOrigin,215.90,-70.47,-0.00),v40,fine,tcp\WObj:=Plywood;
    MoveL Offs(pOrigin,215.90,-70.47,-6.00),v60,z5,tcp\WObj:=Plywood;
    MoveL Offs(pOrigin,214.45,-69.22,-6.00),vTravel,z5,tcp\WObj:=Plywood;
    MoveL Offs(pOrigin,214.45,-69.22,-0.00),v60,z0,tcp\WObj:=Plywood;
    MoveL Offs(pOrigin,213.55,-68.03,-0.00),v40,z0,tcp\WObj:=Plywood;
    MoveL Offs(pOrigin,214.10,-68.03,-0.00),v40,z0,tcp\WObj:=Plywood;
    MoveL Offs(pOrigin,214.55,-69.07,-0.00),v40,z0,tcp\WObj:=Plywood;
    MoveL Offs(pOrigin,215.00,-68.47,-0.00),v40,z0,tcp\WObj:=Plywood;
    MoveL Offs(pOrigin,214.55,-67.72,-0.00),v40,z0,tcp\WObj:=Plywood;
    MoveL Offs(pOrigin,213.80,-67.32,-0.00),v40,z0,tcp\WObj:=Plywood;
    MoveL Offs(pOrigin,212.75,-67.72,-0.00),v40,z0,tcp\WObj:=Plywood;
    MoveL Offs(pOrigin,212.20,-68.78,-0.00),v40,z0,tcp\WObj:=Plywood;
    MoveL Offs(pOrigin,212.45,-69.68,-0.00),v40,z0,tcp\WObj:=Plywood;
    MoveL Offs(pOrigin,213.35,-70.12,-0.00),v40,z0,tcp\WObj:=Plywood;
    MoveL Offs(pOrigin,213.95,-69.97,-0.00),v40,z0,tcp\WObj:=Plywood;
    MoveL Offs(pOrigin,214.45,-69.22,-0.00),v40,z0,tcp\WObj:=Plywood;
    MoveL Offs(pOrigin,213.45,-69.18,-0.00),v40,z0,tcp\WObj:=Plywood;
    MoveL Offs(pOrigin,213.10,-69.18,-0.00),v40,z0,tcp\WObj:=Plywood;
    MoveL Offs(pOrigin,212.95,-68.68,-0.00),v40,z0,tcp\WObj:=Plywood;
    MoveL Offs(pOrigin,213.45,-69.18,-0.00),v40,fine,tcp\WObj:=Plywood;
    MoveL Offs(pOrigin,213.45,-69.18,-6.00),v60,z5,tcp\WObj:=Plywood;
    MoveL Offs(pOrigin,211.40,-68.93,-6.00),vTravel,z5,tcp\WObj:=Plywood;
    MoveL Offs(pOrigin,211.40,-68.93,-0.00),v60,z0,tcp\WObj:=Plywood;
    MoveL Offs(pOrigin,213.15,-66.68,-0.00),v40,z0,tcp\WObj:=Plywood;
    MoveL Offs(pOrigin,212.75,-66.57,-0.00),v40,z0,tcp\WObj:=Plywood;
    MoveL Offs(pOrigin,210.65,-68.47,-0.00),v40,z0,tcp\WObj:=Plywood;
    MoveL Offs(pOrigin,210.55,-68.93,-0.00),v40,z0,tcp\WObj:=Plywood;
    MoveL Offs(pOrigin,211.40,-68.93,-0.00),v40,fine,tcp\WObj:=Plywood;
    MoveL Offs(pOrigin,211.40,-68.93,-6.00),v60,z5,tcp\WObj:=Plywood;
    MoveL Offs(pOrigin,211.25,-67.38,-6.00),vTravel,z5,tcp\WObj:=Plywood;
    MoveL Offs(pOrigin,211.25,-67.38,-0.00),v60,z0,tcp\WObj:=Plywood;
    MoveL Offs(pOrigin,211.50,-66.97,-0.00),v40,z0,tcp\WObj:=Plywood;
    MoveL Offs(pOrigin,210.60,-66.53,-0.00),v40,z0,tcp\WObj:=Plywood;
    MoveL Offs(pOrigin,210.55,-65.78,-0.00),v40,z0,tcp\WObj:=Plywood;
    MoveL Offs(pOrigin,211.85,-65.28,-0.00),v40,z0,tcp\WObj:=Plywood;
    MoveL Offs(pOrigin,211.70,-64.93,-0.00),v40,z0,tcp\WObj:=Plywood;
    MoveL Offs(pOrigin,210.95,-64.97,-0.00),v40,z0,tcp\WObj:=Plywood;
    MoveL Offs(pOrigin,209.95,-65.93,-0.00),v40,z0,tcp\WObj:=Plywood;
    MoveL Offs(pOrigin,210.15,-66.82,-0.00),v40,z0,tcp\WObj:=Plywood;
    MoveL Offs(pOrigin,210.65,-67.32,-0.00),v40,z0,tcp\WObj:=Plywood;
    MoveL Offs(pOrigin,211.25,-67.38,-0.00),v40,fine,tcp\WObj:=Plywood;
    MoveL Offs(pOrigin,211.25,-67.38,-6.00),v60,z5,tcp\WObj:=Plywood;
    MoveL Offs(pOrigin,212.30,-66.32,-6.00),vTravel,z5,tcp\WObj:=Plywood;
    MoveL Offs(pOrigin,212.30,-66.32,-0.00),v60,z0,tcp\WObj:=Plywood;
    MoveL Offs(pOrigin,212.50,-65.93,-0.00),v40,z0,tcp\WObj:=Plywood;
    MoveL Offs(pOrigin,212.15,-65.43,-0.00),v40,z0,tcp\WObj:=Plywood;
    MoveL Offs(pOrigin,212.00,-66.07,-0.00),v40,z0,tcp\WObj:=Plywood;
    MoveL Offs(pOrigin,212.30,-66.32,-0.00),v40,fine,tcp\WObj:=Plywood;
    MoveL Offs(pOrigin,212.30,-66.32,-6.00),v60,z5,tcp\WObj:=Plywood;
    MoveL Offs(pOrigin,202.75,-107.07,-6.00),vTravel,z5,tcp\WObj:=Plywood;
    MoveL Offs(pOrigin,202.75,-107.07,-0.00),v60,z0,tcp\WObj:=Plywood;
    MoveL Offs(pOrigin,203.15,-108.03,-0.00),v40,z0,tcp\WObj:=Plywood;
    MoveL Offs(pOrigin,202.80,-107.93,-0.00),v40,z0,tcp\WObj:=Plywood;
    MoveL Offs(pOrigin,202.75,-107.07,-0.00),v40,fine,tcp\WObj:=Plywood;
    MoveL Offs(pOrigin,202.75,-107.07,-6.00),v60,z5,tcp\WObj:=Plywood;
    MoveL Offs(pOrigin,204.50,-108.43,-6.00),vTravel,z5,tcp\WObj:=Plywood;
    MoveL Offs(pOrigin,204.50,-108.43,-0.00),v60,z0,tcp\WObj:=Plywood;
    MoveL Offs(pOrigin,202.85,-110.03,-0.00),v40,z0,tcp\WObj:=Plywood;
    MoveL Offs(pOrigin,203.00,-110.47,-0.00),v40,z0,tcp\WObj:=Plywood;
    MoveL Offs(pOrigin,204.35,-111.38,-0.00),v40,z0,tcp\WObj:=Plywood;
    MoveL Offs(pOrigin,206.00,-109.72,-0.00),v40,z0,tcp\WObj:=Plywood;
    MoveL Offs(pOrigin,205.70,-109.47,-0.00),v40,z0,tcp\WObj:=Plywood;
    MoveL Offs(pOrigin,204.05,-110.57,-0.00),v40,z0,tcp\WObj:=Plywood;
    MoveL Offs(pOrigin,203.95,-109.88,-0.00),v40,z0,tcp\WObj:=Plywood;
    MoveL Offs(pOrigin,204.75,-108.82,-0.00),v40,z0,tcp\WObj:=Plywood;
    MoveL Offs(pOrigin,204.50,-108.43,-0.00),v40,fine,tcp\WObj:=Plywood;
    MoveL Offs(pOrigin,204.50,-108.43,-6.00),v60,z5,tcp\WObj:=Plywood;
    MoveL Offs(pOrigin,206.30,-110.18,-6.00),vTravel,z5,tcp\WObj:=Plywood;
    MoveL Offs(pOrigin,206.30,-110.18,-0.00),v60,z0,tcp\WObj:=Plywood;
    MoveL Offs(pOrigin,204.80,-111.68,-0.00),v40,z0,tcp\WObj:=Plywood;
    MoveL Offs(pOrigin,205.85,-113.07,-0.00),v40,z0,tcp\WObj:=Plywood;
    MoveL Offs(pOrigin,206.75,-113.12,-0.00),v40,z0,tcp\WObj:=Plywood;
    MoveL Offs(pOrigin,207.55,-112.43,-0.00),v40,z0,tcp\WObj:=Plywood;
    MoveL Offs(pOrigin,207.60,-111.38,-0.00),v40,z0,tcp\WObj:=Plywood;
    MoveL Offs(pOrigin,206.95,-110.62,-0.00),v40,z0,tcp\WObj:=Plywood;
    MoveL Offs(pOrigin,207.20,-109.78,-0.00),v40,z0,tcp\WObj:=Plywood;
    MoveL Offs(pOrigin,206.30,-110.18,-0.00),v40,fine,tcp\WObj:=Plywood;
    MoveL Offs(pOrigin,206.30,-110.18,-6.00),v60,z5,tcp\WObj:=Plywood;
    MoveL Offs(pOrigin,206.00,-111.38,-6.00),vTravel,z5,tcp\WObj:=Plywood;
    MoveL Offs(pOrigin,206.00,-111.38,-0.00),v60,z0,tcp\WObj:=Plywood;
    MoveL Offs(pOrigin,207.05,-111.38,-0.00),v40,z0,tcp\WObj:=Plywood;
    MoveL Offs(pOrigin,207.20,-111.68,-0.00),v40,z0,tcp\WObj:=Plywood;
    MoveL Offs(pOrigin,206.75,-112.43,-0.00),v40,z0,tcp\WObj:=Plywood;
    MoveL Offs(pOrigin,205.85,-112.43,-0.00),v40,z0,tcp\WObj:=Plywood;
    MoveL Offs(pOrigin,206.00,-111.38,-0.00),v40,fine,tcp\WObj:=Plywood;
    MoveL Offs(pOrigin,206.00,-111.38,-6.00),v60,z5,tcp\WObj:=Plywood;
    MoveL Offs(pOrigin,206.65,-113.62,-6.00),vTravel,z5,tcp\WObj:=Plywood;
    MoveL Offs(pOrigin,206.65,-113.62,-0.00),v60,z0,tcp\WObj:=Plywood;
    MoveL Offs(pOrigin,207.20,-114.38,-0.00),v40,z0,tcp\WObj:=Plywood;
    MoveL Offs(pOrigin,207.45,-114.38,-0.00),v40,z0,tcp\WObj:=Plywood;
    MoveL Offs(pOrigin,208.25,-112.32,-0.00),v40,z0,tcp\WObj:=Plywood;
    MoveL Offs(pOrigin,206.65,-113.62,-0.00),v40,z0,tcp\WObj:=Plywood;
    MoveL Offs(pOrigin,207.50,-114.43,-0.00),v40,z0,tcp\WObj:=Plywood;
    MoveL Offs(pOrigin,207.50,-114.68,-0.00),v40,z0,tcp\WObj:=Plywood;
    MoveL Offs(pOrigin,208.25,-114.93,-0.00),v40,z0,tcp\WObj:=Plywood;
    MoveL Offs(pOrigin,209.55,-113.47,-0.00),v40,z0,tcp\WObj:=Plywood;
    MoveL Offs(pOrigin,208.25,-114.32,-0.00),v40,z0,tcp\WObj:=Plywood;
    MoveL Offs(pOrigin,207.50,-114.43,-0.00),v40,fine,tcp\WObj:=Plywood;
    MoveL Offs(pOrigin,207.50,-114.43,-6.00),v60,z5,tcp\WObj:=Plywood;
    MoveL Offs(pOrigin,208.85,-115.57,-6.00),vTravel,z5,tcp\WObj:=Plywood;
    MoveL Offs(pOrigin,208.85,-115.57,-0.00),v60,z0,tcp\WObj:=Plywood;
    MoveL Offs(pOrigin,209.00,-116.18,-0.00),v40,z0,tcp\WObj:=Plywood;
    MoveL Offs(pOrigin,209.25,-116.18,-0.00),v40,z0,tcp\WObj:=Plywood;
    MoveL Offs(pOrigin,209.45,-115.12,-0.00),v40,z0,tcp\WObj:=Plywood;
  ENDPROC

  PROC DrawPart16()
    MoveL Offs(pOrigin,210.20,-114.43,-0.00),v40,z0,tcp\WObj:=Plywood;
    MoveL Offs(pOrigin,209.30,-114.68,-0.00),v40,z0,tcp\WObj:=Plywood;
    MoveL Offs(pOrigin,208.85,-115.57,-0.00),v40,fine,tcp\WObj:=Plywood;
    MoveL Offs(pOrigin,208.85,-115.57,-6.00),v60,z5,tcp\WObj:=Plywood;
    MoveL Offs(pOrigin,209.95,-116.47,-6.00),vTravel,z5,tcp\WObj:=Plywood;
    MoveL Offs(pOrigin,209.95,-116.47,-0.00),v60,z0,tcp\WObj:=Plywood;
    MoveL Offs(pOrigin,210.05,-116.88,-0.00),v40,z0,tcp\WObj:=Plywood;
    MoveL Offs(pOrigin,210.45,-116.32,-0.00),v40,z0,tcp\WObj:=Plywood;
    MoveL Offs(pOrigin,209.95,-116.47,-0.00),v40,z0,tcp\WObj:=Plywood;
    MoveL Offs(pOrigin,210.80,-115.72,-0.00),v40,z0,tcp\WObj:=Plywood;
    MoveL Offs(pOrigin,211.10,-115.88,-0.00),v40,z0,tcp\WObj:=Plywood;
    MoveL Offs(pOrigin,211.25,-115.57,-0.00),v40,z0,tcp\WObj:=Plywood;
    MoveL Offs(pOrigin,210.80,-115.72,-0.00),v40,z0,tcp\WObj:=Plywood;
    MoveL Offs(pOrigin,211.10,-115.88,-0.00),v40,z0,tcp\WObj:=Plywood;
    MoveL Offs(pOrigin,211.10,-115.43,-0.00),v40,z0,tcp\WObj:=Plywood;
    MoveL Offs(pOrigin,210.80,-115.72,-0.00),v40,fine,tcp\WObj:=Plywood;
    MoveL Offs(pOrigin,210.80,-115.72,-6.00),v60,z5,tcp\WObj:=Plywood;
    MoveL Offs(pOrigin,199.10,-115.12,-6.00),vTravel,z5,tcp\WObj:=Plywood;
    MoveL Offs(pOrigin,199.10,-115.12,-0.00),v60,z0,tcp\WObj:=Plywood;
    MoveL Offs(pOrigin,198.80,-113.78,-0.00),v40,z0,tcp\WObj:=Plywood;
    MoveL Offs(pOrigin,197.90,-113.32,-0.00),v40,z0,tcp\WObj:=Plywood;
    MoveL Offs(pOrigin,197.50,-113.78,-0.00),v40,z0,tcp\WObj:=Plywood;
    MoveL Offs(pOrigin,198.45,-114.38,-0.00),v40,z0,tcp\WObj:=Plywood;
    MoveL Offs(pOrigin,198.50,-114.82,-0.00),v40,z0,tcp\WObj:=Plywood;
    MoveL Offs(pOrigin,197.15,-114.07,-0.00),v40,z0,tcp\WObj:=Plywood;
    MoveL Offs(pOrigin,196.40,-114.53,-0.00),v40,z0,tcp\WObj:=Plywood;
    MoveL Offs(pOrigin,195.80,-115.43,-0.00),v40,z0,tcp\WObj:=Plywood;
    MoveL Offs(pOrigin,196.10,-116.32,-0.00),v40,z0,tcp\WObj:=Plywood;
    MoveL Offs(pOrigin,197.00,-117.03,-0.00),v40,z0,tcp\WObj:=Plywood;
    MoveL Offs(pOrigin,198.50,-116.03,-0.00),v40,z0,tcp\WObj:=Plywood;
    MoveL Offs(pOrigin,199.10,-115.12,-0.00),v40,fine,tcp\WObj:=Plywood;
    MoveL Offs(pOrigin,199.10,-115.12,-6.00),v60,z5,tcp\WObj:=Plywood;
    MoveL Offs(pOrigin,197.80,-115.57,-6.00),vTravel,z5,tcp\WObj:=Plywood;
    MoveL Offs(pOrigin,197.80,-115.57,-0.00),v60,z0,tcp\WObj:=Plywood;
    MoveL Offs(pOrigin,197.15,-116.22,-0.00),v40,z0,tcp\WObj:=Plywood;
    MoveL Offs(pOrigin,196.70,-116.22,-0.00),v40,z0,tcp\WObj:=Plywood;
    MoveL Offs(pOrigin,196.65,-115.43,-0.00),v40,z0,tcp\WObj:=Plywood;
    MoveL Offs(pOrigin,197.45,-114.88,-0.00),v40,z0,tcp\WObj:=Plywood;
    MoveL Offs(pOrigin,197.80,-115.57,-0.00),v40,fine,tcp\WObj:=Plywood;
    MoveL Offs(pOrigin,197.80,-115.57,-6.00),v60,z5,tcp\WObj:=Plywood;
    MoveL Offs(pOrigin,195.80,-114.82,-6.00),vTravel,z5,tcp\WObj:=Plywood;
    MoveL Offs(pOrigin,195.80,-114.82,-0.00),v60,z0,tcp\WObj:=Plywood;
    MoveL Offs(pOrigin,196.95,-113.47,-0.00),v40,z0,tcp\WObj:=Plywood;
    MoveL Offs(pOrigin,196.40,-112.82,-0.00),v40,z0,tcp\WObj:=Plywood;
    MoveL Offs(pOrigin,195.35,-114.22,-0.00),v40,z0,tcp\WObj:=Plywood;
    MoveL Offs(pOrigin,194.80,-114.07,-0.00),v40,z0,tcp\WObj:=Plywood;
    MoveL Offs(pOrigin,194.80,-113.62,-0.00),v40,z0,tcp\WObj:=Plywood;
    MoveL Offs(pOrigin,195.80,-112.28,-0.00),v40,z0,tcp\WObj:=Plywood;
    MoveL Offs(pOrigin,195.50,-111.88,-0.00),v40,z0,tcp\WObj:=Plywood;
    MoveL Offs(pOrigin,194.90,-112.12,-0.00),v40,z0,tcp\WObj:=Plywood;
    MoveL Offs(pOrigin,195.00,-111.38,-0.00),v40,z0,tcp\WObj:=Plywood;
    MoveL Offs(pOrigin,194.35,-110.62,-0.00),v40,z0,tcp\WObj:=Plywood;
    MoveL Offs(pOrigin,194.60,-109.43,-0.00),v40,z0,tcp\WObj:=Plywood;
    MoveL Offs(pOrigin,194.00,-109.32,-0.00),v40,z0,tcp\WObj:=Plywood;
    MoveL Offs(pOrigin,192.80,-110.62,-0.00),v40,z0,tcp\WObj:=Plywood;
    MoveL Offs(pOrigin,193.30,-109.88,-0.00),v40,z0,tcp\WObj:=Plywood;
    MoveL Offs(pOrigin,192.80,-109.32,-0.00),v40,z0,tcp\WObj:=Plywood;
    MoveL Offs(pOrigin,191.45,-110.47,-0.00),v40,z0,tcp\WObj:=Plywood;
    MoveL Offs(pOrigin,191.20,-109.88,-0.00),v40,z0,tcp\WObj:=Plywood;
    MoveL Offs(pOrigin,192.00,-108.82,-0.00),v40,z0,tcp\WObj:=Plywood;
    MoveL Offs(pOrigin,192.00,-108.38,-0.00),v40,z0,tcp\WObj:=Plywood;
    MoveL Offs(pOrigin,190.10,-106.53,-0.00),v40,z0,tcp\WObj:=Plywood;
    MoveL Offs(pOrigin,189.20,-106.72,-0.00),v40,z0,tcp\WObj:=Plywood;
    MoveL Offs(pOrigin,188.90,-107.32,-0.00),v40,z0,tcp\WObj:=Plywood;
    MoveL Offs(pOrigin,189.40,-108.53,-0.00),v40,z0,tcp\WObj:=Plywood;
    MoveL Offs(pOrigin,188.45,-107.68,-0.00),v40,z0,tcp\WObj:=Plywood;
    MoveL Offs(pOrigin,188.30,-108.22,-0.00),v40,z0,tcp\WObj:=Plywood;
    MoveL Offs(pOrigin,188.60,-108.97,-0.00),v40,z0,tcp\WObj:=Plywood;
    MoveL Offs(pOrigin,189.65,-109.57,-0.00),v40,z0,tcp\WObj:=Plywood;
    MoveL Offs(pOrigin,190.85,-111.32,-0.00),v40,z0,tcp\WObj:=Plywood;
    MoveL Offs(pOrigin,191.75,-111.38,-0.00),v40,z0,tcp\WObj:=Plywood;
    MoveL Offs(pOrigin,192.30,-111.03,-0.00),v40,z0,tcp\WObj:=Plywood;
    MoveL Offs(pOrigin,191.80,-112.12,-0.00),v40,z0,tcp\WObj:=Plywood;
    MoveL Offs(pOrigin,192.65,-113.07,-0.00),v40,z0,tcp\WObj:=Plywood;
    MoveL Offs(pOrigin,193.95,-113.22,-0.00),v40,z0,tcp\WObj:=Plywood;
    MoveL Offs(pOrigin,193.60,-113.93,-0.00),v40,z0,tcp\WObj:=Plywood;
    MoveL Offs(pOrigin,194.60,-114.97,-0.00),v40,z0,tcp\WObj:=Plywood;
    MoveL Offs(pOrigin,195.20,-115.12,-0.00),v40,z0,tcp\WObj:=Plywood;
    MoveL Offs(pOrigin,195.80,-114.82,-0.00),v40,fine,tcp\WObj:=Plywood;
    MoveL Offs(pOrigin,195.80,-114.82,-6.00),v60,z5,tcp\WObj:=Plywood;
    MoveL Offs(pOrigin,193.85,-112.18,-6.00),vTravel,z5,tcp\WObj:=Plywood;
    MoveL Offs(pOrigin,193.85,-112.18,-0.00),v60,z0,tcp\WObj:=Plywood;
    MoveL Offs(pOrigin,193.00,-112.28,-0.00),v40,z0,tcp\WObj:=Plywood;
    MoveL Offs(pOrigin,193.25,-111.53,-0.00),v40,z0,tcp\WObj:=Plywood;
    MoveL Offs(pOrigin,194.10,-111.53,-0.00),v40,z0,tcp\WObj:=Plywood;
    MoveL Offs(pOrigin,193.85,-112.18,-0.00),v40,fine,tcp\WObj:=Plywood;
    MoveL Offs(pOrigin,193.85,-112.18,-6.00),v60,z5,tcp\WObj:=Plywood;
    MoveL Offs(pOrigin,191.25,-108.43,-6.00),vTravel,z5,tcp\WObj:=Plywood;
    MoveL Offs(pOrigin,191.25,-108.43,-0.00),v60,z0,tcp\WObj:=Plywood;
    MoveL Offs(pOrigin,190.05,-109.38,-0.00),v40,z0,tcp\WObj:=Plywood;
    MoveL Offs(pOrigin,190.70,-108.53,-0.00),v40,z0,tcp\WObj:=Plywood;
    MoveL Offs(pOrigin,191.25,-108.43,-0.00),v40,fine,tcp\WObj:=Plywood;
    MoveL Offs(pOrigin,191.25,-108.43,-6.00),v60,z5,tcp\WObj:=Plywood;
    MoveL Offs(pOrigin,190.05,-108.03,-6.00),vTravel,z5,tcp\WObj:=Plywood;
    MoveL Offs(pOrigin,190.05,-108.03,-0.00),v60,z0,tcp\WObj:=Plywood;
    MoveL Offs(pOrigin,189.80,-107.28,-0.00),v40,z0,tcp\WObj:=Plywood;
    MoveL Offs(pOrigin,190.10,-107.47,-0.00),v40,z0,tcp\WObj:=Plywood;
    MoveL Offs(pOrigin,190.05,-108.03,-0.00),v40,fine,tcp\WObj:=Plywood;
    MoveL Offs(pOrigin,190.05,-108.03,-6.00),v60,z5,tcp\WObj:=Plywood;
    MoveL Offs(pOrigin,188.70,-106.88,-6.00),vTravel,z5,tcp\WObj:=Plywood;
    MoveL Offs(pOrigin,188.70,-106.88,-0.00),v60,z0,tcp\WObj:=Plywood;
    MoveL Offs(pOrigin,187.70,-105.43,-0.00),v40,z0,tcp\WObj:=Plywood;
    MoveL Offs(pOrigin,188.45,-105.68,-0.00),v40,z0,tcp\WObj:=Plywood;
    MoveL Offs(pOrigin,188.75,-106.53,-0.00),v40,z0,tcp\WObj:=Plywood;
    MoveL Offs(pOrigin,189.15,-106.43,-0.00),v40,z0,tcp\WObj:=Plywood;
    MoveL Offs(pOrigin,189.25,-105.82,-0.00),v40,z0,tcp\WObj:=Plywood;
    MoveL Offs(pOrigin,188.30,-104.82,-0.00),v40,z0,tcp\WObj:=Plywood;
    MoveL Offs(pOrigin,186.95,-105.38,-0.00),v40,z0,tcp\WObj:=Plywood;
    MoveL Offs(pOrigin,186.60,-105.97,-0.00),v40,z0,tcp\WObj:=Plywood;
    MoveL Offs(pOrigin,186.60,-106.57,-0.00),v40,z0,tcp\WObj:=Plywood;
    MoveL Offs(pOrigin,187.25,-107.38,-0.00),v40,z0,tcp\WObj:=Plywood;
    MoveL Offs(pOrigin,188.15,-107.38,-0.00),v40,z0,tcp\WObj:=Plywood;
    MoveL Offs(pOrigin,188.70,-106.88,-0.00),v40,z0,tcp\WObj:=Plywood;
    MoveL Offs(pOrigin,187.80,-106.82,-0.00),v40,z0,tcp\WObj:=Plywood;
    MoveL Offs(pOrigin,187.25,-106.72,-0.00),v40,z0,tcp\WObj:=Plywood;
    MoveL Offs(pOrigin,187.15,-106.18,-0.00),v40,z0,tcp\WObj:=Plywood;
    MoveL Offs(pOrigin,187.80,-106.82,-0.00),v40,fine,tcp\WObj:=Plywood;
    MoveL Offs(pOrigin,187.80,-106.82,-6.00),v60,z5,tcp\WObj:=Plywood;
    MoveL Offs(pOrigin,186.35,-105.47,-6.00),vTravel,z5,tcp\WObj:=Plywood;
    MoveL Offs(pOrigin,186.35,-105.47,-0.00),v60,z0,tcp\WObj:=Plywood;
  ENDPROC

  PROC DrawPart17()
    MoveL Offs(pOrigin,187.35,-104.18,-0.00),v40,z0,tcp\WObj:=Plywood;
    MoveL Offs(pOrigin,186.95,-104.18,-0.00),v40,z0,tcp\WObj:=Plywood;
    MoveL Offs(pOrigin,185.50,-105.82,-0.00),v40,z0,tcp\WObj:=Plywood;
    MoveL Offs(pOrigin,186.35,-105.47,-0.00),v40,fine,tcp\WObj:=Plywood;
    MoveL Offs(pOrigin,186.35,-105.47,-6.00),v60,z5,tcp\WObj:=Plywood;
    MoveL Offs(pOrigin,185.30,-106.43,-6.00),vTravel,z5,tcp\WObj:=Plywood;
    MoveL Offs(pOrigin,185.30,-106.43,-0.00),v60,z0,tcp\WObj:=Plywood;
    MoveL Offs(pOrigin,185.30,-105.97,-0.00),v40,z0,tcp\WObj:=Plywood;
    MoveL Offs(pOrigin,185.30,-106.43,-0.00),v40,fine,tcp\WObj:=Plywood;
    MoveL Offs(pOrigin,185.30,-106.43,-6.00),v60,z5,tcp\WObj:=Plywood;
    MoveL Offs(pOrigin,186.50,-103.82,-6.00),vTravel,z5,tcp\WObj:=Plywood;
    MoveL Offs(pOrigin,186.50,-103.82,-0.00),v60,z0,tcp\WObj:=Plywood;
    MoveL Offs(pOrigin,186.65,-103.28,-0.00),v40,z0,tcp\WObj:=Plywood;
    MoveL Offs(pOrigin,186.35,-102.93,-0.00),v40,z0,tcp\WObj:=Plywood;
    MoveL Offs(pOrigin,186.20,-103.57,-0.00),v40,z0,tcp\WObj:=Plywood;
    MoveL Offs(pOrigin,186.50,-103.82,-0.00),v40,fine,tcp\WObj:=Plywood;
    MoveL Offs(pOrigin,186.50,-103.82,-6.00),v60,z5,tcp\WObj:=Plywood;
    MoveL Offs(pOrigin,184.85,-113.78,-6.00),vTravel,z5,tcp\WObj:=Plywood;
    MoveL Offs(pOrigin,184.85,-113.78,-0.00),v60,z0,tcp\WObj:=Plywood;
    MoveL Offs(pOrigin,185.45,-113.78,-0.00),v40,z0,tcp\WObj:=Plywood;
    MoveL Offs(pOrigin,184.85,-113.78,-0.00),v40,z0,tcp\WObj:=Plywood;
    MoveL Offs(pOrigin,185.80,-114.38,-0.00),v40,z0,tcp\WObj:=Plywood;
    MoveL Offs(pOrigin,185.60,-115.07,-0.00),v40,z0,tcp\WObj:=Plywood;
    MoveL Offs(pOrigin,185.15,-115.03,-0.00),v40,z0,tcp\WObj:=Plywood;
    MoveL Offs(pOrigin,185.05,-115.88,-0.00),v40,z0,tcp\WObj:=Plywood;
    MoveL Offs(pOrigin,186.10,-115.12,-0.00),v40,z0,tcp\WObj:=Plywood;
    MoveL Offs(pOrigin,186.05,-114.38,-0.00),v40,z0,tcp\WObj:=Plywood;
    MoveL Offs(pOrigin,185.80,-114.38,-0.00),v40,fine,tcp\WObj:=Plywood;
    MoveL Offs(pOrigin,185.80,-114.38,-6.00),v60,z5,tcp\WObj:=Plywood;
    MoveL Offs(pOrigin,184.55,-116.32,-6.00),vTravel,z5,tcp\WObj:=Plywood;
    MoveL Offs(pOrigin,184.55,-116.32,-0.00),v60,z0,tcp\WObj:=Plywood;
    MoveL Offs(pOrigin,184.25,-116.62,-0.00),v40,z0,tcp\WObj:=Plywood;
    MoveL Offs(pOrigin,184.55,-116.78,-0.00),v40,z0,tcp\WObj:=Plywood;
    MoveL Offs(pOrigin,184.70,-116.47,-0.00),v40,z0,tcp\WObj:=Plywood;
    MoveL Offs(pOrigin,184.40,-116.32,-0.00),v40,z0,tcp\WObj:=Plywood;
    MoveL Offs(pOrigin,184.40,-116.78,-0.00),v40,z0,tcp\WObj:=Plywood;
    MoveL Offs(pOrigin,184.70,-116.62,-0.00),v40,z0,tcp\WObj:=Plywood;
    MoveL Offs(pOrigin,184.55,-116.32,-0.00),v40,fine,tcp\WObj:=Plywood;
    MoveL Offs(pOrigin,184.55,-116.32,-6.00),v60,z5,tcp\WObj:=Plywood;
  ENDPROC

ENDMODULE
